(* IEC 61131-3 sources: plc-mcp/plc_tool/src/plc_tool/scl, 4 files *)

(* ---- temperature_control.st ---- *)
FUNCTION_BLOCK "Temperature_Control"
// 输入变量声明
VAR_INPUT
    ActualTemp      : REAL;    // 实际温度值 (摄氏度)
    SetpointTemp    : REAL;    // 目标温度值 (摄氏度)
    ManualMode      : BOOL;    // 手动模式开关
    ManualOutput    : REAL;    // 手动模式下的输出值 (0-100%)
    Reset          : BOOL;     // 复位信号
    EnableControl  : BOOL;     // 控制使能
END_VAR

// 输出变量声明
VAR_OUTPUT
    HeatingOutput   : REAL;    // 加热器输出 (0-100%)
    HighTempAlarm   : BOOL;    // 高温报警
    LowTempAlarm    : BOOL;    // 低温报警
    SystemStatus    : INT;     // 系统状态代码
END_VAR

// 静态变量声明
VAR
    // PID控制参数
    Kp : REAL := 1.5;         // 比例系数
    Ki : REAL := 0.3;         // 积分系数
    Kd : REAL := 0.1;         // 微分系数

    // 内部变量
    Error           : REAL;    // 温度误差
    IntegralSum     : REAL;    // 积分累加值
    LastError       : REAL;    // 上次误差
    DerivativeTerm  : REAL;    // 微分项

    // 报警设置
    HighTempLimit   : REAL := 85.0;    // 高温报警阈值
    LowTempLimit    : REAL := 5.0;     // 低温报警阈值

    // 定时器
    SampleTime      : TIME := T#100MS;  // 采样时间
    Timer           : TON;              // 定时器实例

    // 数据处理
    TempHistory     : ARRAY[0..9] OF REAL;  // 温度历史数据
    HistoryIndex    : INT := 0;             // 历史数据索引
    AverageTemp     : REAL;                 // 平均温度
END_VAR

BEGIN
    // 系统使能检查
    IF NOT EnableControl THEN
        HeatingOutput := 0.0;
        SystemStatus := 0;  // 系统停止
        RETURN;
    END_IF;

    // 复位处理
    IF Reset THEN
        IntegralSum := 0.0;
        LastError := 0.0;
        HeatingOutput := 0.0;
        HistoryIndex := 0;
        SystemStatus := 1;  // 系统复位
        RETURN;
    END_IF;

    // 定时器控制
    Timer(IN := TRUE, PT := SampleTime);
    IF NOT Timer.Q THEN
        RETURN;
    END_IF;
    Timer(IN := FALSE);

    // 温度历史记录更新
    TempHistory[HistoryIndex] := ActualTemp;
    HistoryIndex := (HistoryIndex + 1) MOD 10;

    // 计算平均温度
    AverageTemp := 0.0;
    FOR i := 0 TO 9 DO
        AverageTemp := AverageTemp + TempHistory[i];
    END_FOR;
    AverageTemp := AverageTemp / 10.0;

    // 报警检查
    HighTempAlarm := ActualTemp >= HighTempLimit;
    LowTempAlarm := ActualTemp <= LowTempLimit;

    // 手动/自动模式控制
    IF ManualMode THEN
        HeatingOutput := LIMIT(0.0, ManualOutput, 100.0);
        SystemStatus := 2;  // 手动模式
    ELSE
        // PID控制计算
        Error := SetpointTemp - ActualTemp;

        // 积分项计算
        IntegralSum := IntegralSum + (Error * DINT_TO_REAL(SampleTime) / 1000.0);
        IntegralSum := LIMIT(-100.0, IntegralSum, 100.0);

        // 微分项计算
        DerivativeTerm := (Error - LastError) / (DINT_TO_REAL(SampleTime) / 1000.0);
        LastError := Error;

        // PID输出计算
        HeatingOutput := (Kp * Error) + (Ki * IntegralSum) + (Kd * DerivativeTerm);
        HeatingOutput := LIMIT(0.0, HeatingOutput, 100.0);

        SystemStatus := 3;  // 自动模式
    END_IF;

    // 报警状态更新系统状态
    IF HighTempAlarm OR LowTempAlarm THEN
        SystemStatus := 4;  // 报警状态
    END_IF;

END_FUNCTION_BLOCK

(* ---- fb_example.st ---- *)
VAR_INPUT
    Input1 : BOOL;    // 输入布尔值
    Input2 : INT;     // 输入整数值
END_VAR

VAR_OUTPUT
    Output1 : BOOL;   // 输出布尔值
    Output2 : INT;    // 输出整数值
END_VAR

VAR
    TempVar : REAL;   // 临时变量
END_VAR

BEGIN
    // 简单的示例逻辑
    IF Input1 THEN
        Output1 := TRUE;
        Output2 := Input2 * 2;
    ELSE
        Output1 := FALSE;
        Output2 := Input2;
    END_IF;
END_PROGRAM

(* ---- fb_motor_control.st ---- *)
VAR_INPUT
    Start : BOOL;         // 启动信号
    Stop : BOOL;         // 停止信号
    Speed_SP : REAL;     // 速度设定值 (0-100%)
    Emergency_Stop : BOOL; // 紧急停止
END_VAR

VAR_OUTPUT
    Motor_Running : BOOL;  // 电机运行状态
    Current_Speed : REAL;  // 当前速度
    Error : BOOL;         // 错误状态
    Error_Code : INT;     // 错误代码
END_VAR

VAR
    Motor_State : INT;     // 电机状态 (0:停止, 1:启动中, 2:运行中, 3:停止中, 4:错误)
    Acceleration : REAL;   // 加速度
    Deceleration : REAL;  // 减速度
    Timer : TON;          // 定时器
END_VAR

BEGIN
    // 紧急停止处理
    IF Emergency_Stop THEN
        Motor_State := 4;
        Error := TRUE;
        Error_Code := 1; // 紧急停止错误代码
        Motor_Running := FALSE;
        Current_Speed := 0.0;
        RETURN;
    END_IF;

    // 状态机处理
    CASE Motor_State OF
        0:  // 停止状态
            IF Start AND NOT Stop THEN
                Motor_State := 1;
                Error := FALSE;
                Error_Code := 0;
            END_IF;
            Current_Speed := 0.0;
            Motor_Running := FALSE;

        1:  // 启动中
            Motor_Running := TRUE;
            IF Current_Speed < Speed_SP THEN
                Current_Speed := Current_Speed + Acceleration;
            ELSE
                Motor_State := 2;
            END_IF;

        2:  // 运行中
            IF Stop OR NOT Start THEN
                Motor_State := 3;
            ELSE
                Current_Speed := Speed_SP;
            END_IF;

        3:  // 停止中
            IF Current_Speed > 0.0 THEN
                Current_Speed := Current_Speed - Deceleration;
            ELSE
                Motor_State := 0;
                Motor_Running := FALSE;
            END_IF;

        4:  // 错误状态
            IF NOT Emergency_Stop AND NOT Start THEN
                Motor_State := 0;
                Error := FALSE;
                Error_Code := 0;
            END_IF;
    END_CASE;

    // 限制速度范围
    IF Current_Speed < 0.0 THEN
        Current_Speed := 0.0;
    ELSIF Current_Speed > 100.0 THEN
        Current_Speed := 100.0;
    END_IF;
END_PROGRAM

(* ---- fb_pid_control.st ---- *)
VAR_INPUT
    SetPoint : REAL;      // 设定值
    ActualValue : REAL;   // 实际值
    Kp : REAL;           // 比例系数
    Ki : REAL;           // 积分系数
    Kd : REAL;           // 微分系数
    Enable : BOOL;       // 使能信号
    Reset : BOOL;        // 复位信号
END_VAR

VAR_OUTPUT
    Output : REAL;       // 输出值
    Error : REAL;        // 误差
    Running : BOOL;      // 运行状态
END_VAR

VAR
    Integral : REAL;     // 积分值
    LastError : REAL;    // 上次误差
    DeltaTime : REAL;    // 采样时间
    FirstScan : BOOL;    // 首次扫描标志
END_VAR

BEGIN
    // 初始化
    IF FirstScan THEN
        FirstScan := FALSE;
        DeltaTime := 0.1; // 100ms采样时间
        Integral := 0.0;
        LastError := 0.0;
    END_IF;

    // PID控制
    IF Enable THEN
        Running := TRUE;

        // 计算误差
        Error := SetPoint - ActualValue;

        // 复位处理
        IF Reset THEN
            Integral := 0.0;
            LastError := 0.0;
            Output := 0.0;
            RETURN;
        END_IF;

        // PID算法
        Integral := Integral + Error * DeltaTime;

        // 计算输出
        Output := Kp * Error +                    // 比例项
                 Ki * Integral +                  // 积分项
                 Kd * (Error - LastError) / DeltaTime;  // 微分项

        // 更新上次误差
        LastError := Error;

        // 限制输出范围 (0-100%)
        IF Output < 0.0 THEN
            Output := 0.0;
            Integral := Integral - Error * DeltaTime; // 抗积分饱和
        ELSIF Output > 100.0 THEN
            Output := 100.0;
            Integral := Integral - Error * DeltaTime; // 抗积分饱和
        END_IF;

    ELSE
        Running := FALSE;
        Output := 0.0;
        Integral := 0.0;
        LastError := 0.0;
    END_IF;
END_PROGRAM
